FUNCTION_BLOCK fbWordToReal
VAR_INPUT
	in_B0					: BYTE ;
	in_B1					: BYTE ;
	in_r_Res				: REAL ;
	in_i_Offset				: INT ;
END_VAR
VAR_OUTPUT
	out_r_Value				: REAL ;
END_VAR
VAR
	dw_AddedValue			: DWORD;
	r_ResolutionResolved	: REAL;
END_VAR

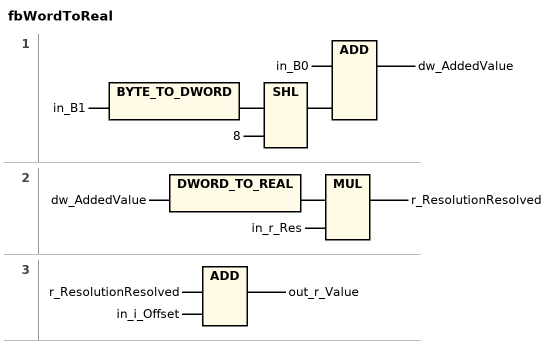
// NETWORK 1
dw_AddedValue := in_B0 + SHL(BYTE_TO_DWORD(in_B1), 8);

// NETWORK 2
r_ResolutionResolved := DWORD_TO_REAL(dw_AddedValue) * in_r_Res;

// NETWORK 3
out_r_Value := r_ResolutionResolved + in_i_Offset;

END_FUNCTION_BLOCK

(* stored: Version 1.1.0.1, ProductVersion 3.1.4024.12
   POU fbWordToReal: Id {c451e33c-33f6-44a2-b1bc-a55c49d6a6c5}, SpecialFunc None *)
